TYPE "pnioSubnetStatus"
TITLE = {"version":"v1.0","author":"cyanezf","family":"core/fieldbus/pnio-diag","status":"current","deprecatedBy": null,"dependencies":["pnioDeviceStatus-v1.0"]}

//(*--
//# Documentation
//## Log
//| version | date | author | description |
//|:-------:|:----:|:------:|:------------|
//| v1.0 | 2022-10-12 | cyanezf | First version |
//
//## Description
//PNIO subnet status
//--*)

   STRUCT
      state : Int;   // Current state
      error : Int;   // Current error
      device { S7_SetPoint := 'False'} : Array[0..1023] of "pnioDeviceStatus";   // Devices
   END_STRUCT;

END_TYPE

